Staubli VAL3: onF8Event.pgx

program onF8Event(bool& l_bSave[])
  local num x_nResult
begin
  // look if the bButton is enable
  if bButton[7]
    //
    call saveIt(l_bSave)
  endIf
end
